// Mitsubishi GX Developer project: Automatic-Doors-GX-Mitshubishi-PLC   PLC: FX2N

PROGRAM MAIN
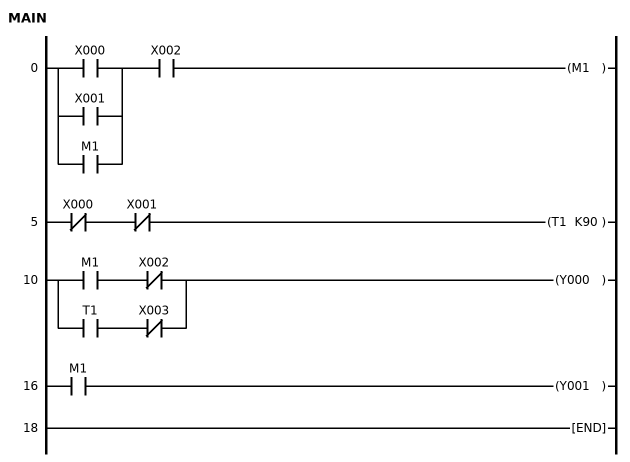
0     LD      X000
      OR      X001
      OR      M1
      AND     X002
      OUT     M1
5     LDI     X000
      ANI     X001
      OUT     T1 K90
10    LD      M1
      ANI     X002
      LD      T1
      ANI     X003
      ORB
      OUT     Y000
16    LD      M1
      OUT     Y001
18    END
END_PROGRAM
